Staubli VAL3: setEnable.pgx

public program setEnable(bool x_bEnable, string x_sItem)
  local num l_nSize
begin
  // check if is active
  saveInOut:dOutput[x_sItem].bEnable=x_bEnable
end
